// TIA Portal V20 export
TYPE "typeCmControlNodeInterlock"
// stored: Namespace Unit1.Em3
   STRUCT
      topTapeAxisX : "LER_typeAxisInterlock";
      topTapeAxisY : "LER_typeAxisInterlock";
      topTapeLoading : "LER_typeTwoWayActuatorInterlock";
      topTapeLoadingClamp : "LER_typeTwoWayActuatorInterlock";
      topTapeCutterUpDown : "LER_typeTwoWayActuatorInterlock";
      topTapeCutterClamp : "LER_typeTwoWayActuatorInterlock";
      topTapeTension : "LER_typeTwoWayActuatorInterlock";
      topTapeAttachment : "LER_typeTwoWayActuatorInterlock";
      topTapeClampTopLeft : "LER_typeTwoWayActuatorInterlock";
      topTapeClampTopCenter : "LER_typeTwoWayActuatorInterlock";
      topTapeClampTopRight : "LER_typeTwoWayActuatorInterlock";
      topTapeClampBtm : "LER_typeTwoWayActuatorInterlock";
      topTapeClampAll : "LER_typeTwoWayActuatorInterlock";
      topTapeAttachmentVaccum : "LER_typeTwoWayActuatorInterlock";
   END_STRUCT;
END_TYPE
